SUBAPPLICATION Uebung_006_SAFE_AX (* SAFE-Variante: Wiederanlaufsperre fuer Uebung_006_AX (SF_ResetButton, I7/I8) *)
  (* Standard: 61499-2; Description: Copyright (c) 2026 Meisterschulen am Ostbahnhof This program and the accompanying materials are made available under the terms of the Eclipse Public License 2.0 which is available at https://www.eclipse.org/legal/epl-2.0/ SPDX-License-Identifier: EPL-2.0 *)
  (* Version 1.0, 2026-10-09, Franz Höpfinger, Meisterschulen am Ostbahnhof, SAFE-Variante von Uebung_006_AX. STOP (I2) und Meldeeingang I8 (HW-Not-Halt-Rueckmeldung) schalten den Ausgang SW-seitig sofort ab und sperren START per StartPermit-Latch (E_RS) + StartGate (E_PERMIT), bis RESET (I7) ueber SF_ResetButton (PLCopen Safety Part 1 Ch. 6.1) eine gueltige Tasten-Flanke erkennt. RESET alleine schaltet den Ausgang nicht wieder ein, dafuer muss START erneut gedrueckt werden. *)
  PACKAGE Uebungen;
  IMPORT logiBUS::io::DI::logiBUS_DI::Input_I1;
  IMPORT logiBUS::io::DI::logiBUS_DI::Input_I2;
  IMPORT logiBUS::io::DI::logiBUS_DI::Input_I7;
  IMPORT logiBUS::io::DI::logiBUS_DI::Input_I8;
  IMPORT logiBUS::io::DI::logiBUS_DI_Events::BUTTON_SINGLE_CLICK;
  IMPORT logiBUS::io::DI::logiBUS_DI_Events::BUTTON_PRESS_DOWN;
  IMPORT logiBUS::io::DQ::logiBUS_DO::Output_Q1;
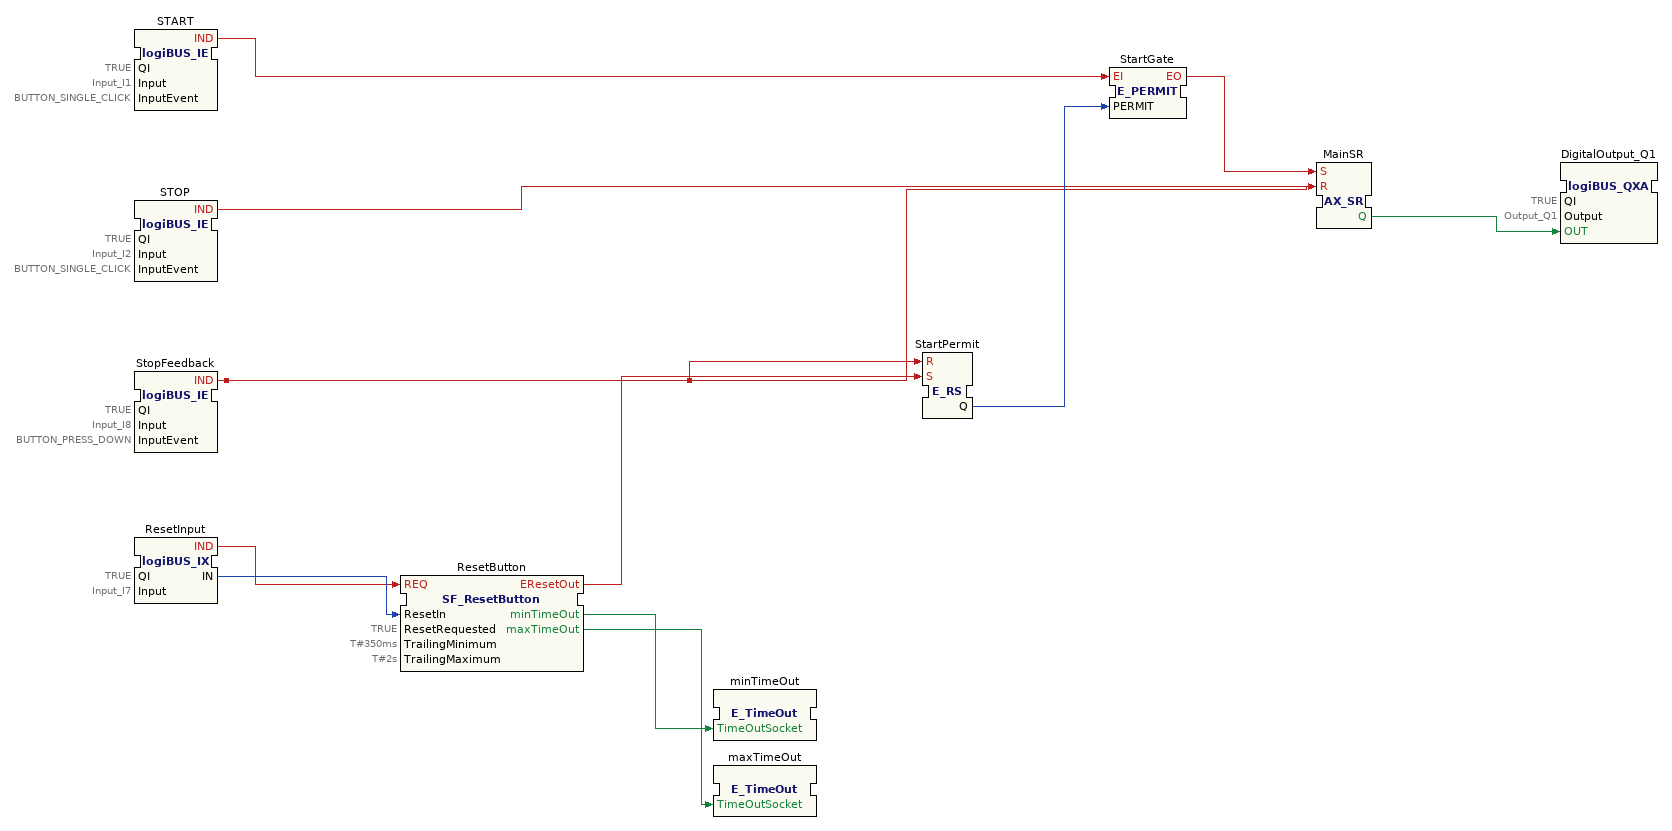
  FBS
    START : logiBUS::io::DI::logiBUS_IE(QI := TRUE, Input := Input_I1, InputEvent := BUTTON_SINGLE_CLICK); (* Taster START *)
    STOP : logiBUS::io::DI::logiBUS_IE(QI := TRUE, Input := Input_I2, InputEvent := BUTTON_SINGLE_CLICK); (* Hand-Stopp (nicht HW-Not-Halt) *)
    StopFeedback : logiBUS::io::DI::logiBUS_IE(QI := TRUE, Input := Input_I8, InputEvent := BUTTON_PRESS_DOWN); (* Meldeeingang HW-Not-Halt *)
    ResetInput : logiBUS::io::DI::logiBUS_IX(QI := TRUE, Input := Input_I7); (* Pegel+Event fuer SF_ResetButton *)
    ResetButton : logiBUS::safety::PLCopen::SF_ResetButton(ResetRequested := TRUE, TrailingMinimum := T#350ms, TrailingMaximum := T#2s);
    StartPermit : iec61499::events::E_RS; (* Freigabe-Latch (E_RS statt E_SR nur wegen kreuzungsfreier Verdrahtung) *)
    StartGate : iec61499::events::E_PERMIT; (* Laesst START nur bei Freigabe durch *)
    MainSR : adapter::events::unidirectional::AX_SR;
    DigitalOutput_Q1 : logiBUS::io::DQ::logiBUS_QXA(QI := TRUE, Output := Output_Q1);
    minTimeOut : iec61499::events::E_TimeOut;
    maxTimeOut : iec61499::events::E_TimeOut;
  END_FBS
  EVENT_CONNECTIONS
    START.IND TO StartGate.EI;
    StartGate.EO TO MainSR.S;
    STOP.IND TO MainSR.R;
    StopFeedback.IND TO MainSR.R;
    StopFeedback.IND TO StartPermit.R;
    ResetInput.IND TO ResetButton.REQ;
    ResetButton.EResetOut TO StartPermit.S;
  END_CONNECTIONS
  DATA_CONNECTIONS
    ResetInput.IN TO ResetButton.ResetIn;
    StartPermit.Q TO StartGate.PERMIT;
  END_CONNECTIONS
  ADAPTER_CONNECTIONS
    MainSR.Q TO DigitalOutput_Q1.OUT;
    ResetButton.minTimeOut TO minTimeOut.TimeOutSocket;
    ResetButton.maxTimeOut TO maxTimeOut.TimeOutSocket;
  END_CONNECTIONS
END_SUBAPPLICATION
